// TwinCAT 3 PLC project Untitled1
// ProgramVersion: 3.1.4024.0
// libraries:
//   Tc2_EtherCAT, * (Beckhoff Automation GmbH)
//   Tc2_MC2, * (Beckhoff Automation GmbH)
//   Tc2_Standard, * (Beckhoff Automation GmbH)
//   Tc2_System, * (Beckhoff Automation GmbH)
//   Tc3_EventLogger, * (Beckhoff Automation GmbH)
//   Tc3_Module, * (Beckhoff Automation GmbH)
// project tree:
//   GVLs/ GVL.TcGVL
//   / PlcTask.TcTTO
//   POUs/ MAIN.TcPOU
// real-time tasks:
//   TASK PlcTask: cycle T#10ms, priority 20, ADS port 350
// motion (NC):
//   TASK NC-Task 1 SAF: cycle T#4ms, priority 4, ADS port 501
//   TASK NC-Task 1 SVB: cycle T#10ms, priority 8, ADS port 511
//   AXIS Axis 1 (id 1)
//     Dynamic: AccelerationMaximum=150000, DecelerationMaximum=150000, Acceleration=5566, Deceleration=5566, Jerk=5566
//     Velo: SlowManual=5000, FastManual=150000, Maximum=150000
//     PositionAreaControl: Enable=false
//     TargetPosControl: Enable=false
//     OtherSettings: AllowMotionCmdToSlave=true
//     encoder EncType=19
//       EncPara: ScaleFactorNumerator=1, MaxCount=#xffffffff
//     drive DrvType=16
//       DrvPara: MaxCount=#xffffffff, DriveControlDWord=#x00020000
//         Analog: VeloReferenz=150000, TorqueSetpointScale=10, ScaleFactorActTorque=0.1
//         TimeComp: TaskDelayCycles=1
//     controller CtrType=1
//       CtrPara: PriorControlFactor=1
//         PosDiffControl: Enable=false
//         Observer: BandWidth=20
// I/O:
//   DEVICE Device 1 (EtherCAT), AmsNetId 192.168.1.160.2.1
//     Drive 1 (ZeroErr Driver) [ZeroErr Driver]
// variable links:
//   NC-Task 1 SAF/Axes/Axis 1 <-> Device 1 (EtherCAT)/Drive 1 (ZeroErr Driver)
//     Drive/Inputs/In/nDcOutputTime <-> InfoData/DcOutputShift
//     Drive/Inputs/In/nState1 <-> Transmit PDO mapping 0/Status word
//     Drive/Inputs/In/nState2 <-> Transmit PDO mapping 0/Status word @bit 8
//     Drive/Inputs/In/nState4 @bit 1 <-> WcState/InputToggle
//     Drive/Inputs/In/nState4 <-> WcState/WcState
//     Drive/Outputs/Out/nCtrl1 <-> Receive PDO mapping 0/Control word
//     Drive/Outputs/Out/nCtrl2 <-> Receive PDO mapping 0/Control word @bit 8
//     Drive/Outputs/Out/nDataOut1 <-> Receive PDO mapping 0/Target Position
//     Drive/Outputs/Out/nDataOut4[0] <-> Receive PDO mapping 0/Target Torque
//     Enc/Inputs/In/nDataIn1 <-> Transmit PDO mapping 0/Position actual value
//     Enc/Inputs/In/nDataIn7 <-> Transmit PDO mapping 0/Actual velocity
//     Enc/Inputs/In/nDcInputTime <-> InfoData/DcInputShift
//     Enc/Inputs/In/nState4 @bit 1 <-> WcState/InputToggle
//     Enc/Inputs/In/nState4 <-> WcState/WcState
//   Untitled1/Untitled1 Instance <-> Device 1 (EtherCAT)/Drive 1 (ZeroErr Driver)
//     PlcTask Inputs/GVL.Actual_Position <-> Transmit PDO mapping 0/Position actual value_1
//     PlcTask Inputs/GVL.Actual_Velocity <-> Transmit PDO mapping 0/Actual velocity_1
//     PlcTask Outputs/GVL.Operation_Mode <-> Receive PDO mapping 0/Modes of operation
//     PlcTask Outputs/GVL.Profile_acceleration <-> Receive PDO mapping 0/Profile acceleration
//     PlcTask Outputs/GVL.Profile_deceleration <-> Receive PDO mapping 0/Profile deceleration
//     PlcTask Outputs/GVL.Target_Velocity <-> Receive PDO mapping 0/Target Velocity
//   Untitled1/Untitled1 Instance <-> NC-Task 1 SAF/Axes/Axis 1
//     PlcTask Inputs/MAIN.axis1.NcToPlc <-> Outputs/ToPlc
//     PlcTask Outputs/MAIN.axis1.PlcToNc <-> Inputs/FromPlc

CONFIGURATION Untitled1
    RESOURCE PLC ON TwinCAT3
        TASK PlcTask(INTERVAL := T#10ms, PRIORITY := 20);
        PROGRAM MAIN WITH PlcTask : MAIN;
    END_RESOURCE
END_CONFIGURATION

// ---- GVLs/GVL.TcGVL
{attribute 'qualified_only'}
VAR_GLOBAL
	Actual_Velocity   AT%I*   :DINT ;
	Actual_Position   AT%I*   :DINT ;

	Control_word      AT%Q*   :INT  :=  0;
	Target_Velocity   AT%Q*   :DINT  := 0;	
	Target_Position   AT%Q*   :DINT  := 0;
	Operation_Mode    AT%Q*   :SINT  := 0;
	Profile_acceleration			  AT%Q*   :DINT  := 0;
	Profile_deceleration		      AT%Q*   :DINT  := 0;
END_VAR

// ---- POUs/MAIN.TcPOU
PROGRAM MAIN
VAR
    (* 功能块 *)
    axis1: AXIS_REF;    (* 轴引用 *)

    (* 功能块 *)
    MCPower : MC_Power; (* 电机上电/下电控制功能块 *)
    MCJog   : MC_Jog;   (* 点动控制功能块 *)
	fbMoveCyclicPosition :MC_MoveRelative;
    fbMoveAbs      : MC_MoveAbsolute; // 定义绝对位置运动功能块
	MC_JOG :MC_JOG;


END_VAR

(* 使用速度控制 

*)

MCPower(Enable := TRUE,
		Enable_Positive := TRUE,
		Enable_Negative := TRUE,
		Override := 100,
		Axis  := axis1,
);
// 运动到绝对位置


//fbMoveCyclicPosition(Axis := axis1,Execute := TRUE, Distance:=3000,Velocity := 3000);

END_PROGRAM
